Omron Sysmac Studio project node_red_nx1p2_MODUL (Sysmac Studio 1.47.0.64008, StandardProject)

# Controller new_Controller_0: NX1P2-9024DT version 1.40
Units and slaves: Node86 : NX-ECC201 (E001); Unit 1 : NX-OD5121 (N1); Unit 2 : NX-OD4256 (N2); Unit 3 : NX-ID5342 (N3); Unit 4 : NX-ID5442 (N4); Node1 : GX-ID1611+OD16 (E002)
Task PrimaryTask (priority 4, period or condition 2000): Program0

VAR_GLOBAL RETAIN
    SETPOINT AT %D5 : INT;  (* published *)
    A1 AT %D7 : INT;  (* published *)
    VALUE AT %D8 : INT;
    CONTROL_OUT_1 AT %D9 : INT;  (* published *)
    CONTROL_OUT_2 AT %D10 : INT;  (* published *)
    CONTROL_OUT_0_OD4256 AT %D30 : INT;  (* CONTROL_OD4256_IO; published *)
END_VAR
VAR_GLOBAL
    OUT_1 : BOOL;  (* at BuiltInIO://cpu/#0/Output_Bit_00 *)
    OUT_2 : BOOL;  (* at BuiltInIO://cpu/#0/Output_Bit_01 *)
END_VAR
VAR_GLOBAL RETAIN
    CONTROL_OUT_1_OD4256 AT %D31 : INT;  (* CONTROL_OD4256_IO; published *)
    CONTROL_OUT_2_OD4256 AT %D32 : INT;  (* CONTROL_OD4256_IO; published *)
    CONTROL_OUT_3_OD4256 AT %D33 : INT;  (* CONTROL_OD4256_IO; published *)
    CONTROL_OUT_4_OD4256 AT %D34 : INT;  (* CONTROL_OD4256_IO; published *)
    CONTROL_OUT_5_OD4256 AT %D35 : INT;  (* CONTROL_OD4256_IO; published *)
    CONTROL_OUT_6_OD4256 AT %D36 : INT;  (* CONTROL_OD4256_IO; published *)
    CONTROL_OUT_7_OD4256 AT %D37 : INT;  (* CONTROL_OD4256_IO; published *)
    CONTROL_OUT_0_OD5121 AT %D40 : INT;  (* CONTROL_OD4256_IO; published *)
    CONTROL_OUT_1_OD5121 AT %D41 : INT;  (* CONTROL_OD4256_IO; published *)
    CONTROL_OUT_2_OD5121 AT %D42 : INT;  (* CONTROL_OD4256_IO; published *)
    CONTROL_OUT_3_OD5121 AT %D43 : INT;  (* CONTROL_OD4256_IO; published *)
    CONTROL_OUT_4_OD5121 AT %D44 : INT;  (* CONTROL_OD4256_IO; published *)
    CONTROL_OUT_5_OD5121 AT %D45 : INT;  (* CONTROL_OD4256_IO; published *)
    CONTROL_OUT_6_OD5121 AT %D46 : INT;  (* CONTROL_OD4256_IO; published *)
    CONTROL_OUT_7_OD5121 AT %D47 : INT;  (* CONTROL_OD4256_IO; published *)
    CONTROL_OUT_8_OD5121 AT %D48 : INT;  (* CONTROL_OD4256_IO; published *)
    CONTROL_OUT_9_OD5121 AT %D49 : INT;  (* CONTROL_OD4256_IO; published *)
    CONTROL_OUT_10_OD5121 AT %D10 : INT;  (* CONTROL_OD4256_IO; published *)
    CONTROL_OUT_11_OD5121 AT %D51 : INT;  (* CONTROL_OD4256_IO; published *)
    CONTROL_OUT_12_OD5121 AT %D52 : INT;  (* CONTROL_OD4256_IO; published *)
    CONTROL_OUT_13_OD5121 AT %D53 : INT;  (* CONTROL_OD4256_IO; published *)
    CONTROL_OUT_14_OD5121 AT %D54 : INT;  (* CONTROL_OD4256_IO; published *)
    CONTROL_OUT_15_OD5121 AT %D55 : INT;  (* CONTROL_OD4256_IO; published *)
END_VAR
VAR_GLOBAL
    OD4256_OUT_0 : BOOL;  (* at ECAT://node#[86,2]/Output Bit 8 bits/Output Bit 00 *)
    OD4256_OUT_1 : BOOL;  (* at ECAT://node#[86,2]/Output Bit 8 bits/Output Bit 01 *)
    OD4256_OUT_2 : BOOL;  (* at ECAT://node#[86,2]/Output Bit 8 bits/Output Bit 02 *)
    OD4256_OUT_3 : BOOL;  (* at ECAT://node#[86,2]/Output Bit 8 bits/Output Bit 03 *)
    OD4256_OUT_4 : BOOL;  (* at ECAT://node#[86,2]/Output Bit 8 bits/Output Bit 04 *)
    OD4256_OUT_5 : BOOL;  (* at ECAT://node#[86,2]/Output Bit 8 bits/Output Bit 05 *)
    OD4256_OUT_6 : BOOL;  (* at ECAT://node#[86,2]/Output Bit 8 bits/Output Bit 06 *)
    OD4256_OUT_7 : BOOL;  (* at ECAT://node#[86,2]/Output Bit 8 bits/Output Bit 07 *)
    OD5121_OUT_0 : BOOL;  (* at ECAT://node#[86,1]/Output Bit 16 bits/Output Bit 00 *)
    OD5121_OUT_1 : BOOL;  (* at ECAT://node#[86,1]/Output Bit 16 bits/Output Bit 01 *)
    OD5121_OUT_2 : BOOL;  (* at ECAT://node#[86,1]/Output Bit 16 bits/Output Bit 02 *)
END_VAR

PROGRAM Program0
VAR
    Timer_1 : BOOL;
    timer_a1 : TON;
    T : TIME;
    C : INT;
END_VAR
VAR_EXTERNAL
    A1 : INT;
    VALUE : INT;
    SETPOINT : INT;
    CONTROL_OUT_1 : INT;
    OUT_1 : BOOL;
    CONTROL_OUT_2 : INT;
    OUT_2 : BOOL;
    CONTROL_OUT_0_OD4256 : INT;
    OD4256_OUT_0 : BOOL;
    CONTROL_OUT_1_OD4256 : INT;
    OD4256_OUT_1 : BOOL;
    CONTROL_OUT_2_OD4256 : INT;
    OD4256_OUT_2 : BOOL;
    CONTROL_OUT_3_OD4256 : INT;
    OD4256_OUT_3 : BOOL;
    CONTROL_OUT_4_OD4256 : INT;
    OD4256_OUT_4 : BOOL;
    CONTROL_OUT_5_OD4256 : INT;
    OD4256_OUT_5 : BOOL;
    CONTROL_OUT_6_OD4256 : INT;
    OD4256_OUT_6 : BOOL;
    CONTROL_OUT_7_OD4256 : INT;
    OD4256_OUT_7 : BOOL;
    CONTROL_OUT_0_OD5121 : INT;
    OD5121_OUT_0 : BOOL;
    CONTROL_OUT_1_OD5121 : INT;
    OD5121_OUT_1 : BOOL;
    CONTROL_OUT_2_OD5121 : INT;
    OD5121_OUT_2 : BOOL;
END_VAR
VAR
    _e1 : R_TRIG;
END_VAR

(* Section Section0: ladder, written here as Structured Text *)

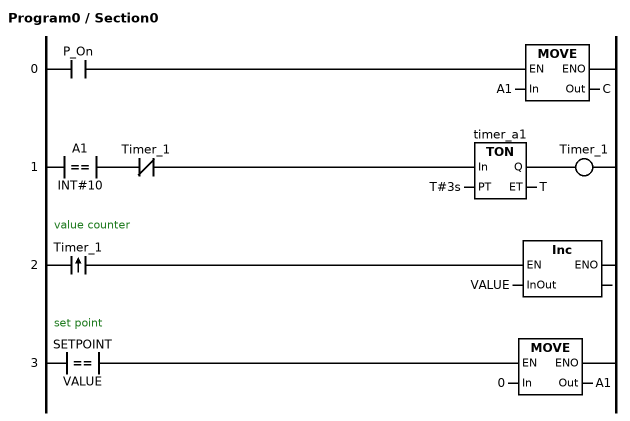
(* Rung 0 *)
IF P_On THEN C := A1; END_IF;
(* Rung 1 *)
timer_a1(In := (A1 = INT#10) AND NOT Timer_1, PT := T#3s, ET => T);
Timer_1 := timer_a1.Q;
(* Rung 2: value counter *)
_e1(CLK := Timer_1);
IF _e1.Q THEN Inc(InOut := VALUE); END_IF;
(* Rung 3: set point *)
IF SETPOINT = VALUE THEN A1 := 0; END_IF;

(* Section remote_io: ladder, written here as Structured Text *)

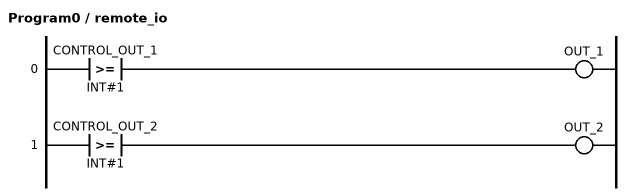
(* Rung 0 *)
OUT_1 := CONTROL_OUT_1 >= INT#1;
(* Rung 1 *)
OUT_2 := CONTROL_OUT_2 >= INT#1;

(* Section CONTROL_OD4256: ladder, written here as Structured Text *)

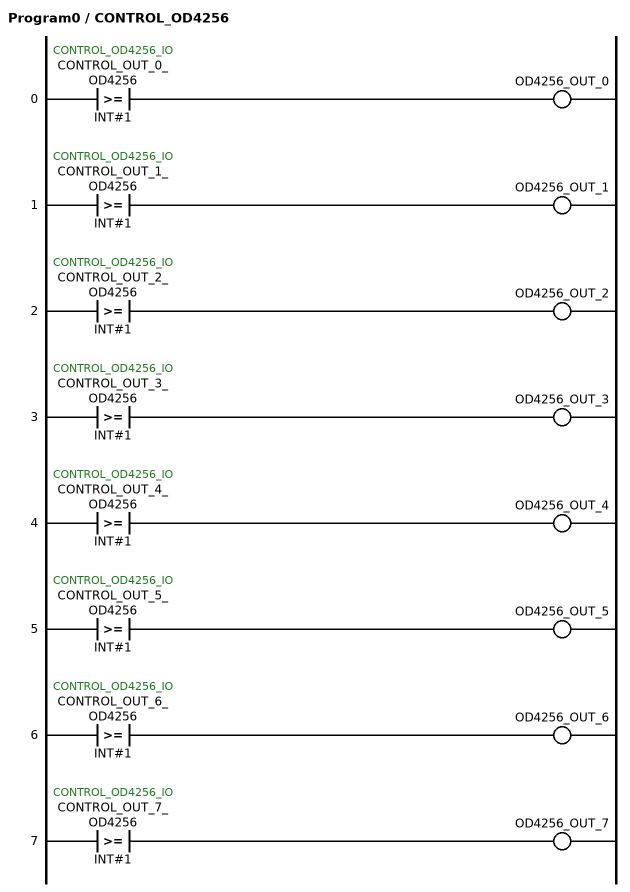
(* Rung 0 *)
OD4256_OUT_0 := CONTROL_OUT_0_OD4256 >= INT#1;
(* Rung 1 *)
OD4256_OUT_1 := CONTROL_OUT_1_OD4256 >= INT#1;
(* Rung 2 *)
OD4256_OUT_2 := CONTROL_OUT_2_OD4256 >= INT#1;
(* Rung 3 *)
OD4256_OUT_3 := CONTROL_OUT_3_OD4256 >= INT#1;
(* Rung 4 *)
OD4256_OUT_4 := CONTROL_OUT_4_OD4256 >= INT#1;
(* Rung 5 *)
OD4256_OUT_5 := CONTROL_OUT_5_OD4256 >= INT#1;
(* Rung 6 *)
OD4256_OUT_6 := CONTROL_OUT_6_OD4256 >= INT#1;
(* Rung 7 *)
OD4256_OUT_7 := CONTROL_OUT_7_OD4256 >= INT#1;

(* Section CONTROL_OD5121: ladder, written here as Structured Text *)

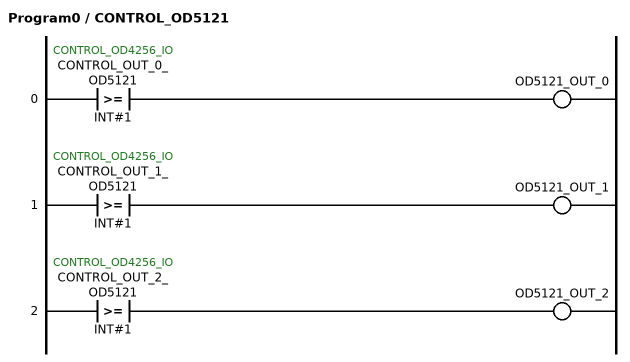
(* Rung 0 *)
OD5121_OUT_0 := CONTROL_OUT_0_OD5121 >= INT#1;
(* Rung 1 *)
OD5121_OUT_1 := CONTROL_OUT_1_OD5121 >= INT#1;
(* Rung 2 *)
OD5121_OUT_2 := CONTROL_OUT_2_OD5121 >= INT#1;
END_PROGRAM